(* PLC project mapp1, BrAutomation SafeDESIGNER  6.0.0.2 *)
(* stored: companyURL http://www.br-automation.com, creationDateTime Tue Oct 01 11:48:23 2024 *)

PROGRAM Main

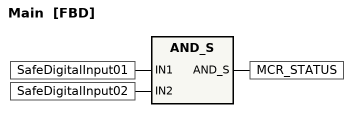
(* FBD diagram, written out as Structured Text *)
MCR_STATUS := AND_S(SafeDigitalInput01, SafeDigitalInput02);
END_PROGRAM
